FUNCTION_BLOCK tetsssssssssssztsgzdazigaeuof
VAR_INPUT
END_VAR
VAR_OUTPUT
END_VAR
VAR
END_VAR

END_FUNCTION_BLOCK

(* stored: Version 1.1.0.1, ProductVersion 3.1.4026.12
   POU tetsssssssssssztsgzdazigaeuof: Id {18fcae89-dd34-4cc6-8f9f-401e193fe429}, SpecialFunc None *)
